// TIA Portal V19 export
TYPE "typeAOPD_Function"
// Safety status of light curtain
// stored: Access Published, IsFailsafeCompliant true, Namespace Safety
   STRUCT
      released { ExternalWritable := 'False'} : Bool;   // Curtain OK
      ackReq { ExternalWritable := 'False'} : Bool;   // Acknowledge required
   END_STRUCT;
END_TYPE
